(* CODESYS project Tarea_automa.project

Project tree, tasks and I/O mapping:
  Device : CODESYS Control Win V3, 3S - Smart Software Solutions GmbH, order no. 305021, version 3.5.7.20
    application Application
      libraries: Standard, * (System); Util, * (System)
      task MainTask (cyclic, interval t#20ms, priority 1) calls PLC_PRG
      program PLC_PRG [FBD]
      global variables GVL
*)

// Device/Application/GVL
VAR_GLOBAL
	PV: REAL;
	SP: REAL;
END_VAR

// Device/Application/PLC_PRG
PROGRAM PLC_PRG
VAR
	PID_H: PID;
END_VAR

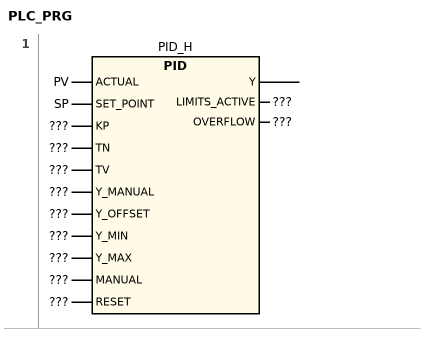
// NETWORK 1
PID_H(ACTUAL := PV, SET_POINT := SP); // PID

END_PROGRAM
